{attribute 'qualified_only'}
VAR_GLOBAL
	b_StartAuto : BOOL;
	b_StopAuto : BOOL;
	ProgramSelect : DINT;
END_VAR

(* stored: Version 1.1.0.1
   GVL GVL_HMI: Id {17a5de81-b901-449a-9fc1-ca9aa50e1960} *)
